PROGRAM POU
VAR
END_VAR

END_PROGRAM

(* stored: Version 1.1.0.1, ProductVersion 3.1.4024.12
   POU POU: Id {2bff8c3f-40fc-4dbb-be99-2995d31e7b3b}, SpecialFunc None *)
